PROGRAM MAIN
VAR
END_VAR

MotionControl();

END_PROGRAM

(* stored: Version 1.1.0.1, ProductVersion 3.1.4024.9
   POU MAIN: Id {45d3f657-a2aa-4170-8e90-2d1edb6d9fbd}, SpecialFunc None *)
